// TIA Portal V19 export
FUNCTION "Peeler_CALL" : Void   // FC119, LAD
TITLE = LOWER PEELER & SNUBBER MACHINE CALL
// stored: SetENOAutomatically false
BEGIN

REGION Network 1: Data In - PB
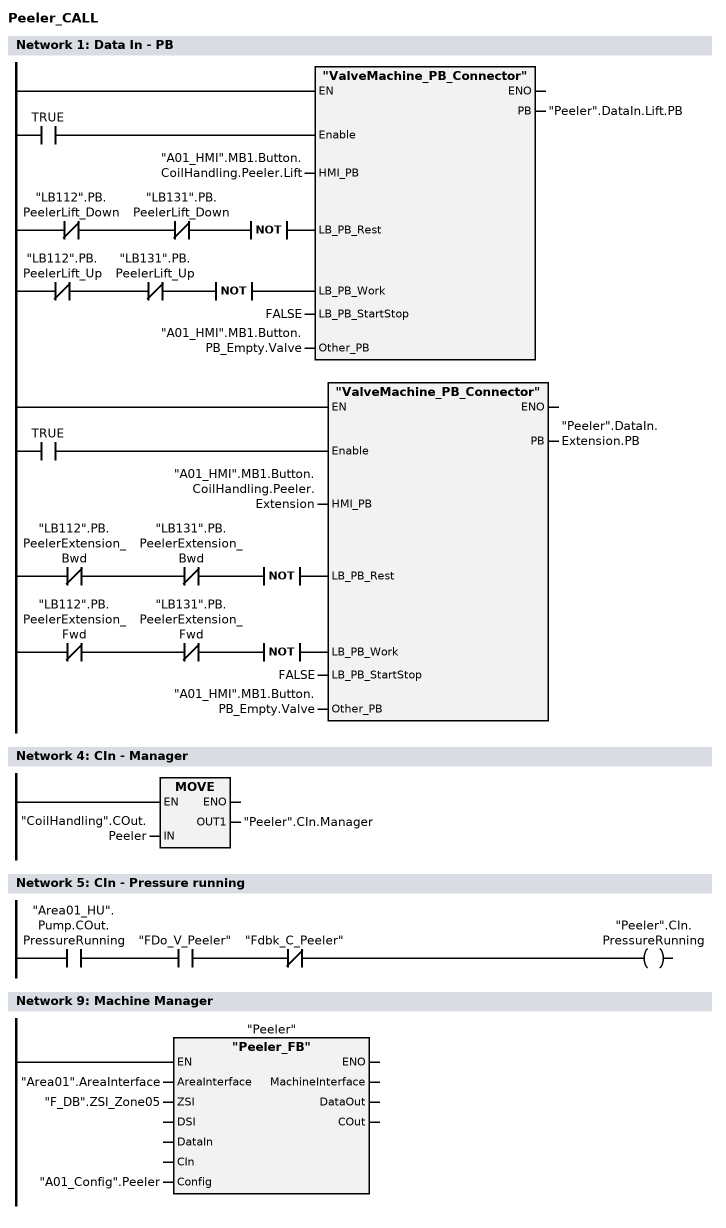
   RUNG wire#powerrail
      "ValveMachine_PB_Connector"(Enable := wire#w1, LB_PB_Rest := wire#w2, LB_PB_Work := wire#w3, HMI_PB := "A01_HMI".MB1.Button.CoilHandling.Peeler.Lift, LB_PB_StartStop := FALSE, Other_PB := "A01_HMI".MB1.Button.PB_Empty.Valve, PB => "Peeler".DataIn.Lift.PB)
   END_RUNG
   RUNG wire#powerrail
      Contact( TRUE )
   END_RUNG wire#w1
   RUNG wire#powerrail
      I_Contact( "LB112".PB.PeelerLift_Down )
      I_Contact( "LB131".PB.PeelerLift_Down )
      Not()
   END_RUNG wire#w2
   RUNG wire#powerrail
      I_Contact( "LB112".PB.PeelerLift_Up )
      I_Contact( "LB131".PB.PeelerLift_Up )
      Not()
   END_RUNG wire#w3
   RUNG wire#powerrail
      "ValveMachine_PB_Connector"(Enable := wire#w4, LB_PB_Rest := wire#w5, LB_PB_Work := wire#w6, HMI_PB := "A01_HMI".MB1.Button.CoilHandling.Peeler.Extension, LB_PB_StartStop := FALSE, Other_PB := "A01_HMI".MB1.Button.PB_Empty.Valve, PB => "Peeler".DataIn.Extension.PB)
   END_RUNG
   RUNG wire#powerrail
      Contact( TRUE )
   END_RUNG wire#w4
   RUNG wire#powerrail
      I_Contact( "LB112".PB.PeelerExtension_Bwd )
      I_Contact( "LB131".PB.PeelerExtension_Bwd )
      Not()
   END_RUNG wire#w5
   RUNG wire#powerrail
      I_Contact( "LB112".PB.PeelerExtension_Fwd )
      I_Contact( "LB131".PB.PeelerExtension_Fwd )
      Not()
   END_RUNG wire#w6
   // the same network as SCL:
   "ValveMachine_PB_Connector"(Enable := TRUE,
                           HMI_PB := "A01_HMI".MB1.Button.CoilHandling.Peeler.Lift,
                           LB_PB_Rest := NOT (NOT "LB112".PB.PeelerLift_Down AND NOT "LB131".PB.PeelerLift_Down),
                           LB_PB_Work := NOT (NOT "LB112".PB.PeelerLift_Up AND NOT "LB131".PB.PeelerLift_Up),
                           LB_PB_StartStop := FALSE,
                           Other_PB := "A01_HMI".MB1.Button.PB_Empty.Valve,
                           PB => "Peeler".DataIn.Lift.PB);
   "ValveMachine_PB_Connector"(Enable := TRUE,
                           HMI_PB := "A01_HMI".MB1.Button.CoilHandling.Peeler.Extension,
                           LB_PB_Rest := NOT (NOT "LB112".PB.PeelerExtension_Bwd AND NOT "LB131".PB.PeelerExtension_Bwd),
                           LB_PB_Work := NOT (NOT "LB112".PB.PeelerExtension_Fwd AND NOT "LB131".PB.PeelerExtension_Fwd),
                           LB_PB_StartStop := FALSE,
                           Other_PB := "A01_HMI".MB1.Button.PB_Empty.Valve,
                           PB => "Peeler".DataIn.Extension.PB);
END_REGION

REGION Network 2 (SCL): DataIn - Sensors
   //Lift
   //
   "Peeler".DataIn.Lift.Rest_Ls[1] := "Peeler_Ls_Down";
   "Peeler".DataIn.Lift.Work_Ls[1] := "Peeler_Ls_Up";

   // Extension
   // 
   "Peeler".DataIn.Extension.Rest_Ls[1] := "Peeler_Ls_Bwd";
   "Peeler".DataIn.Extension.Work_Ls[1] := FALSE; //"Peeler_Ls_Fwd"; NON ESISTE
END_REGION

REGION Network 3: >
END_REGION

REGION Network 4: CIn - Manager
   RUNG wire#powerrail
      Move(in := "CoilHandling".COut.Peeler, out1 => "Peeler".CIn.Manager)
   END_RUNG
   // the same network as SCL:
   "Peeler".CIn.Manager := "CoilHandling".COut.Peeler;
END_REGION

REGION Network 5: CIn - Pressure running
   RUNG wire#powerrail
      Contact( "Area01_HU".Pump.COut.PressureRunning )
      Contact( "FDo_V_Peeler" )
      I_Contact( "Fdbk_C_Peeler" )
      Coil( "Peeler".CIn.PressureRunning )
   END_RUNG
   // the same network as SCL:
   "Peeler".CIn.PressureRunning := "Area01_HU".Pump.COut.PressureRunning AND "FDo_V_Peeler" AND NOT "Fdbk_C_Peeler";
END_REGION

REGION Network 6: >
END_REGION

REGION Network 7 (SCL): DSI
   "Peeler".DSI.Extension :=
   "Peeler".DSI.LIft := "F_DB".DSI_V_Peeler;
END_REGION

REGION Network 8: >
END_REGION

REGION Network 9: Machine Manager
   RUNG wire#powerrail
      "Peeler"(AreaInterface := "Area01".AreaInterface, ZSI := "F_DB".ZSI_Zone05, DSI :=, DataIn :=, CIn :=, Config := "A01_Config".Peeler, MachineInterface =>, DataOut =>, COut =>)
   END_RUNG
   // the same network as SCL:
   "Peeler"(AreaInterface := "Area01".AreaInterface, ZSI := "F_DB".ZSI_Zone05, Config := "A01_Config".Peeler);   // "Peeler_FB"
END_REGION

REGION Network 10: >
END_REGION

REGION Network 11 (SCL): Data Out
   // Lift
   // 
   "Peeler_V_Down" := "Peeler".DataOut.Lift.RestSolenoid;
   "Peeler_V_Up" := "Peeler".DataOut.Lift.WorkSolenoid;

   // Extension
   // 
   "Peeler_V_Bwd" := "Peeler".DataOut.Extension.RestSolenoid;
   "Peeler_V_Fwd" := "Peeler".DataOut.Extension.WorkSolenoid;
END_REGION

REGION Network 12: >
END_REGION
END_FUNCTION
